// TIA Portal V20 export
VAR_GLOBAL   // PLC tag table "Default tag table"
   Tag_1 AT %M1.0 : Bool;
END_VAR
